Staubli VAL3: stop.pgx

program stop()
begin
//*******************************************************************************
//*   ______
//*  / _____) /|
//* | |      / /
//* | | /\  / /
//* | | \ \/ /  _      Copyright (c) KEOLABS, 2016
//* | |  \__/  | |        http://www.keolabs.com
//* | |________| |
//*  \__________/
//*
//********************************************************************************
//*@file          : start
//*@author        : Yves Ragot
//*@version       : $Id: stop.pgx 1176 2016-10-03 15:44:15Z yves $
//*@brief         : stop program of Rob6x
//*
  //*******************************************************************************/

  call KillAllTasks()

end
